(* CoDeSys 2.3.9.28 project: muj kolotoc.pro *)
(* Libraries: Standard.lib 2.12.10 14:48:34, SYSLIBCALLBACK.LIB 2.12.10 14:48:32 *)

(* PLC configuration (modules and I/O channels)
K-Bus [K_Bus] node 0, in %IB0 out %QB0
Fieldbus variables [FB_VARS] node 1, in %IB0 out %QB0
Flag variables [FLAG_VARS] node 2, in %IB0 out %QB0
*)

(* POU PLC_PRG, CFC *)
PROGRAM PLC_PRG
VAR
	Plus: BOOL;
	Minus: BOOL;
	a: BOOL;
	b: BOOL;
	c: BOOL;
	d: BOOL;
	e: BOOL;
	f: BOOL;
	g: BOOL;
	h: BOOL;
	ch: BOOL;
	i: BOOL;
	kolotoc: KolotocF;
END_VAR
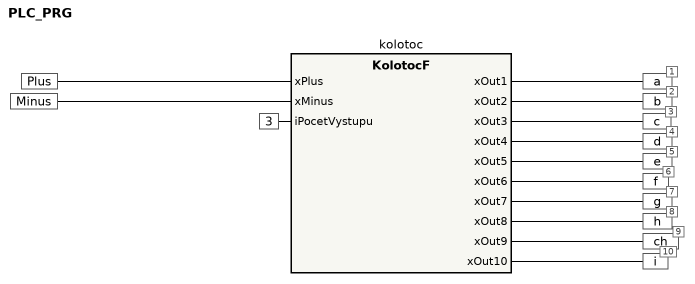
_CFC_ (* Continuous Function Chart, elements in execution order *)
#0 kolotoc:KolotocF(xPlus: Plus, xMinus: Minus, iPocetVystupu: 3)
#1 a <= #0.xOut1
#2 b <= #0.xOut2
#3 c <= #0.xOut3
#4 d <= #0.xOut4
#5 e <= #0.xOut5
#6 f <= #0.xOut6
#7 g <= #0.xOut7
#8 h <= #0.xOut8
#9 ch <= #0.xOut9
#10 i <= #0.xOut10
_END_CFC_
(* the same logic as Structured Text *)
kolotoc(xPlus := Plus, xMinus := Minus, iPocetVystupu := 3);
a := kolotoc.xOut1;
b := kolotoc.xOut2;
c := kolotoc.xOut3;
d := kolotoc.xOut4;
e := kolotoc.xOut5;
f := kolotoc.xOut6;
g := kolotoc.xOut7;
h := kolotoc.xOut8;
ch := kolotoc.xOut9;
i := kolotoc.xOut10;
END_PROGRAM

(* POU Kolotoc, ST *)
PROGRAM Kolotoc
VAR
	index: INT := 0;
	a: BOOL := FALSE;
	b: BOOL := FALSE;
END_VAR
VAR_INPUT
	KratkyStiskPlus: BOOL;
	KratkyStiskMinus: BOOL;
	DlouhyStiskPlus: BOOL;
	DlouhyStiskMinus: BOOL;
	PocetAktivnichVystupu: INT;
END_VAR
VAR_OUTPUT
	Rele1: BOOL;
	Rele2: BOOL;
	Rele3: BOOL;
	Rele4: BOOL;
	Rele5: BOOL;
	Rele6: BOOL;
	Rele7: BOOL;
	Rele8: BOOL;
	Rele9: BOOL;
	Rele10: BOOL;
END_VAR
IF (KratkyStiskPlus)
THEN
	a := TRUE;
END_IF

IF (a AND KratkyStiskPlus = FALSE)
	THEN
	index := index + 1;
	a := FALSE;
END_IF

IF (KratkyStiskMinus)
THEN
	b := TRUE;
END_IF

IF (b AND KratkyStiskMinus = FALSE)
THEN
	index := index - 1;
	b := FALSE;
END_IF

IF (index = -1)
THEN
	index := PocetAktivnichVystupu;
END_IF

IF (index = PocetAktivnichVystupu + 1)
THEN
	index := 0;
END_IF

IF (index = 0 )
THEN
	Rele1 := FALSE;
	Rele2 := FALSE;
	Rele3 := FALSE;
	Rele4 := FALSE;
	Rele5 := FALSE;
	Rele6 := FALSE;
	Rele7 := FALSE;
	Rele8 := FALSE;
	Rele9 := FALSE;
	Rele10 := FALSE;
ELSIF (index = 1)
THEN
	Rele1 := TRUE;
	Rele2 := FALSE;
	Rele3 := FALSE;
	Rele4 := FALSE;
	Rele5 := FALSE;
	Rele6 := FALSE;
	Rele7 := FALSE;
	Rele8 := FALSE;
	Rele9 := FALSE;
	Rele10 := FALSE;
ELSIF (index = 2)
THEN
	Rele1 := FALSE;
	Rele2 := TRUE;
	Rele3 := FALSE;
	Rele4 := FALSE;
	Rele5 := FALSE;
	Rele6 := FALSE;
	Rele7 := FALSE;
	Rele8 := FALSE;
	Rele9 := FALSE;
	Rele10 := FALSE;
ELSIF (index = 3)
THEN
	Rele1 := FALSE;
	Rele2 := FALSE;
	Rele3 := TRUE;
	Rele4 := FALSE;
	Rele5 := FALSE;
	Rele6 := FALSE;
	Rele7 := FALSE;
	Rele8 := FALSE;
	Rele9 := FALSE;
	Rele10 := FALSE;
ELSIF (index = 4)
THEN
	Rele1 := FALSE;
	Rele2 := FALSE;
	Rele3 := FALSE;
	Rele4 := TRUE;
	Rele5 := FALSE;
	Rele6 := FALSE;
	Rele7 := FALSE;
	Rele8 := FALSE;
	Rele9 := FALSE;
	Rele10 := FALSE;
ELSIF (index = 5)
THEN
	Rele1 := FALSE;
	Rele2 := FALSE;
	Rele3 := FALSE;
	Rele4 := FALSE;
	Rele5 := TRUE;
	Rele6 := FALSE;
	Rele7 := FALSE;
	Rele8 := FALSE;
	Rele9 := FALSE;
	Rele10 := FALSE;
ELSIF (index = 6)
THEN
	Rele1 := FALSE;
	Rele2 := FALSE;
	Rele3 := FALSE;
	Rele4 := FALSE;
	Rele5 := FALSE;
	Rele6 := TRUE;
	Rele7 := FALSE;
	Rele8 := FALSE;
	Rele9 := FALSE;
	Rele10 := FALSE;
ELSIF (index = 7)
THEN
	Rele1 := FALSE;
	Rele2 := FALSE;
	Rele3 := FALSE;
	Rele4 := FALSE;
	Rele5 := FALSE;
	Rele6 := FALSE;
	Rele7 := TRUE;
	Rele8 := FALSE;
	Rele9 := FALSE;
	Rele10 := FALSE;
ELSIF (index = 8)
THEN
	Rele1 := FALSE;
	Rele2 := FALSE;
	Rele3 := FALSE;
	Rele4 := FALSE;
	Rele5 := FALSE;
	Rele6 := FALSE;
	Rele7 := FALSE;
	Rele8 := TRUE;
	Rele9 := FALSE;
	Rele10 := FALSE;
ELSIF (index = 9)
THEN
	Rele1 := FALSE;
	Rele2 := FALSE;
	Rele3 := FALSE;
	Rele4 := FALSE;
	Rele5 := FALSE;
	Rele6 := FALSE;
	Rele7 := FALSE;
	Rele8 := FALSE;
	Rele9 := TRUE;
	Rele10 := FALSE;
ELSIF (index = 10)
THEN
	Rele1 := FALSE;
	Rele2 := FALSE;
	Rele3 := FALSE;
	Rele4 := FALSE;
	Rele5 := FALSE;
	Rele6 := FALSE;
	Rele7 := FALSE;
	Rele8 := FALSE;
	Rele9 := FALSE;
	Rele10 := TRUE;
END_IF

IF (DlouhyStiskPlus)
THEN
	index := 0;
END_IF

IF (DlouhyStiskMinus)
THEN
	index := 0;
END_IF
END_PROGRAM

(* POU KolotocF, CFC *)
FUNCTION_BLOCK KolotocF
VAR
END_VAR
VAR_INPUT
	xPlus: BOOL;
	xMinus: BOOL;
	iPocetVystupu: INT;
END_VAR
VAR_OUTPUT
	xOut1: BOOL;
	xOut2: BOOL;
	xOut3: BOOL;
	xOut4: BOOL;
	xOut5: BOOL;
	xOut6: BOOL;
	xOut7: BOOL;
	xOut8: BOOL;
	xOut9: BOOL;
	xOut10: BOOL;
END_VAR
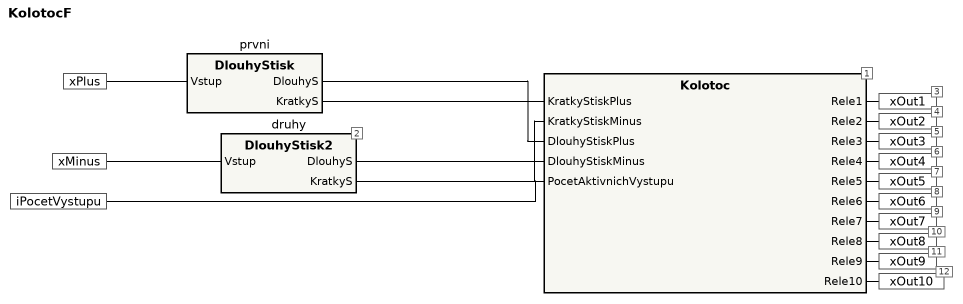
_CFC_ (* Continuous Function Chart, elements in execution order *)
#0 prvni:DlouhyStisk(Vstup: xPlus)
#1 Kolotoc(KratkyStiskPlus: #0.KratkyS, KratkyStiskMinus: #2.KratkyS, DlouhyStiskPlus: #0.DlouhyS, DlouhyStiskMinus: #2.DlouhyS, PocetAktivnichVystupu: iPocetVystupu)
#2 druhy:DlouhyStisk2(Vstup: xMinus)
#3 xOut1 <= #1.Rele1
#4 xOut2 <= #1.Rele2
#5 xOut3 <= #1.Rele3
#6 xOut4 <= #1.Rele4
#7 xOut5 <= #1.Rele5
#8 xOut6 <= #1.Rele6
#9 xOut7 <= #1.Rele7
#10 xOut8 <= #1.Rele8
#11 xOut9 <= #1.Rele9
#12 xOut10 <= #1.Rele10
_END_CFC_
(* the same logic as Structured Text *)
prvni(Vstup := xPlus);
Kolotoc(KratkyStiskPlus := prvni.KratkyS, KratkyStiskMinus := druhy.KratkyS, DlouhyStiskPlus := prvni.DlouhyS, DlouhyStiskMinus := druhy.DlouhyS, PocetAktivnichVystupu := iPocetVystupu);
druhy(Vstup := xMinus);
xOut1 := Kolotoc.Rele1;
xOut2 := Kolotoc.Rele2;
xOut3 := Kolotoc.Rele3;
xOut4 := Kolotoc.Rele4;
xOut5 := Kolotoc.Rele5;
xOut6 := Kolotoc.Rele6;
xOut7 := Kolotoc.Rele7;
xOut8 := Kolotoc.Rele8;
xOut9 := Kolotoc.Rele9;
xOut10 := Kolotoc.Rele10;
END_FUNCTION_BLOCK

(* POU DlouhyStisk, CFC *)
PROGRAM DlouhyStisk
VAR_INPUT
	Vstup: BOOL;
END_VAR
VAR_OUTPUT
	DlouhyS: BOOL;
	KratkyS: BOOL;
END_VAR
VAR
	cas1: TON;
	cas2: TOF;
	cas3: TON;
	cas4: TOF;
END_VAR
VAR (* helpers for the ST form of the networks *)
	_t57 : BOOL;
END_VAR
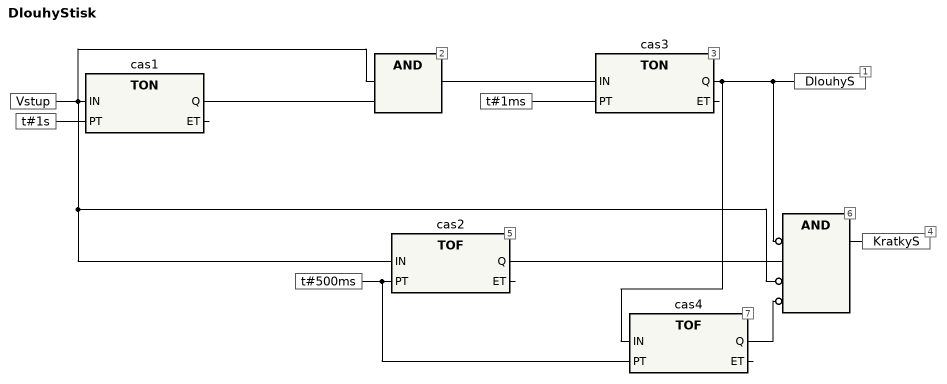
_CFC_ (* Continuous Function Chart, elements in execution order *)
#0 cas1:TON(IN: Vstup, PT: t#1s)
#1 DlouhyS <= #3.Q
#2 AND(Vstup, #0.Q)
#3 cas3:TON(IN: #2, PT: t#1ms)
#4 KratkyS <= #6
#5 cas2:TOF(IN: Vstup, PT: t#500ms)
#6 AND(NOT #3.Q, #5.Q, NOT Vstup, NOT #7.Q)
#7 cas4:TOF(IN: #3.Q, PT: t#500ms)
_END_CFC_
(* the same logic as Structured Text *)
cas1(IN := Vstup, PT := t#1s);
DlouhyS := cas3.Q;
cas3(IN := Vstup AND cas1.Q, PT := t#1ms);
KratkyS := _t57;
cas2(IN := Vstup, PT := t#500ms);
_t57 := NOT cas3.Q AND cas2.Q AND NOT Vstup AND NOT cas4.Q;
cas4(IN := cas3.Q, PT := t#500ms);
END_PROGRAM

(* POU DlouhyStisk2, CFC *)
PROGRAM DlouhyStisk2
VAR_INPUT
	Vstup: BOOL;
END_VAR
VAR_OUTPUT
	DlouhyS: BOOL;
	KratkyS: BOOL;
END_VAR
VAR
	cas1: TON;
	cas2: TOF;
	cas3: TON;
	cas4: TOF;
END_VAR
VAR (* helpers for the ST form of the networks *)
	_t57 : BOOL;
END_VAR
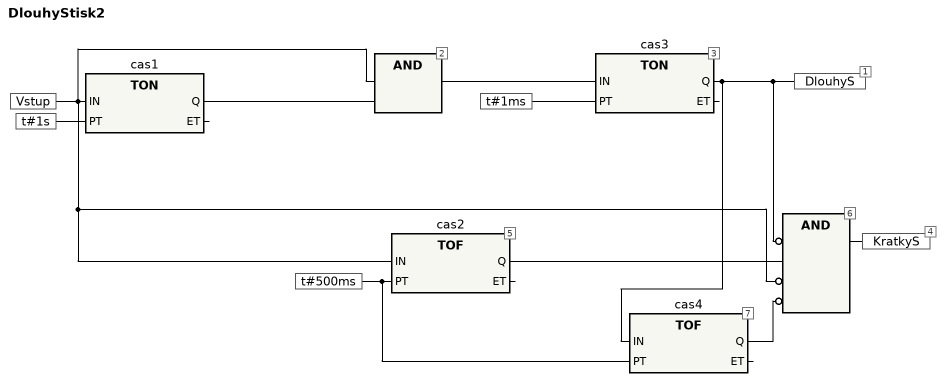
_CFC_ (* Continuous Function Chart, elements in execution order *)
#0 cas1:TON(IN: Vstup, PT: t#1s)
#1 DlouhyS <= #3.Q
#2 AND(Vstup, #0.Q)
#3 cas3:TON(IN: #2, PT: t#1ms)
#4 KratkyS <= #6
#5 cas2:TOF(IN: Vstup, PT: t#500ms)
#6 AND(NOT #3.Q, #5.Q, NOT Vstup, NOT #7.Q)
#7 cas4:TOF(IN: #3.Q, PT: t#500ms)
_END_CFC_
(* the same logic as Structured Text *)
cas1(IN := Vstup, PT := t#1s);
DlouhyS := cas3.Q;
cas3(IN := Vstup AND cas1.Q, PT := t#1ms);
KratkyS := _t57;
cas2(IN := Vstup, PT := t#500ms);
_t57 := NOT cas3.Q AND cas2.Q AND NOT Vstup AND NOT cas4.Q;
cas4(IN := cas3.Q, PT := t#500ms);
END_PROGRAM

(* Visualisation plc_vizu
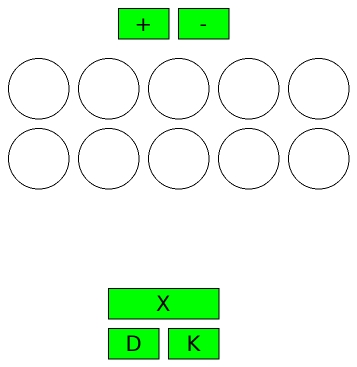
rectangle at (130,10)-(181,41): text "+"; alarm colour if PLC_PRG.Plus; taps PLC_PRG.Plus
rectangle at (190,10)-(241,41): text "-"; alarm colour if PLC_PRG.Minus; taps PLC_PRG.Minus
ellipse at (20,60)-(81,121): alarm colour if PLC_PRG.a
ellipse at (90,60)-(151,121): alarm colour if PLC_PRG.b
ellipse at (160,60)-(221,121): alarm colour if PLC_PRG.c
ellipse at (230,60)-(291,121): alarm colour if PLC_PRG.d
ellipse at (300,60)-(361,121): alarm colour if PLC_PRG.e
ellipse at (20,130)-(81,191): alarm colour if PLC_PRG.f
ellipse at (90,130)-(151,191): alarm colour if PLC_PRG.g
ellipse at (160,130)-(221,191): alarm colour if PLC_PRG.h
ellipse at (230,130)-(291,191): alarm colour if PLC_PRG.ch
ellipse at (300,130)-(361,191): alarm colour if PLC_PRG.i
rectangle at (120,330)-(171,361): text "D"; alarm colour if PLC_PRG.Dlouhy
rectangle at (180,330)-(231,361): text "K"; alarm colour if PLC_PRG.kratky; taps PLC_PRG.kratky
rectangle at (120,290)-(231,321): text "X"; alarm colour if PLC_PRG.x; taps PLC_PRG.x
*)
